FUNCTION rt_ceild : LREAL
VAR_INPUT
	u: LREAL;
END_VAR
VAR
END_VAR


rt_ceild := DINT_TO_LREAL(TRUNC(u));

IF u = rt_ceild THEN 
    rt_ceild := u;
ELSIF u >= 0.0 THEN 
    rt_ceild := rt_ceild + 1.0;
END_IF;

END_FUNCTION

(* stored: Version 1.1.0.1, ProductVersion 3.1.4024.12
   POU rt_ceild: Id {2c546896-7a78-484f-91d6-e0a7f6950c92}, SpecialFunc None *)
